FUNCTION_BLOCK FB_Afstandssensor IMPLEMENTS ITF_Afstandssensor
VAR_INPUT
END_VAR
VAR_OUTPUT
END_VAR
VAR
	// Interne waarden
	Afstand_Intern : LREAL;
	Drempelwaarde_Intern : LREAL;
	
	Detectie_Intern : BOOL;
	Status_Intern : E_AfstandssensorStatus;
END_VAR

PROPERTY Afstand : LREAL
GET
Afstand := Afstand_Intern;
END_GET
SET
VAR
	Waarde : LREAL;
END_VAR
Afstand_Intern := Waarde;
END_SET
END_PROPERTY

PROPERTY Detectie : BOOL
GET
Detectie := Detectie_Intern;
END_GET
END_PROPERTY

PROPERTY Drempelwaarde : LREAL
GET
Drempelwaarde := Drempelwaarde_Intern;
END_GET
SET
VAR
	Waarde : LREAL;
END_VAR
Drempelwaarde_Intern := Waarde;
END_SET
END_PROPERTY

PROPERTY Status : E_AfstandssensorStatus
GET
Status := Status_Intern;
END_GET
END_PROPERTY

METHOD Update : BOOL
// Afstandssensor controleert op interne fouten
IF Afstand_Intern < 0 THEN
	Status_Intern := E_AfstandssensorStatus.Error;
	Detectie_Intern := FALSE;
	RETURN;
END_IF

// Afstandssensor controleert op drempelwaarde
IF Afstand_Intern <= Drempelwaarde_Intern THEN
	Detectie_Intern := TRUE; 
	Status_Intern := E_AfstandssensorStatus.Detectie;
ELSE
	Detectie_Intern := FALSE; 
	Status_Intern := E_AfstandssensorStatus.Normaal;
END_IF
END_METHOD

END_FUNCTION_BLOCK

(* stored: Version 1.1.0.1
   POU FB_Afstandssensor: Id {72d78e64-2ca1-40bf-a72f-434aeebace35}, SpecialFunc None
   Folder Methods: Id {64d0ffcc-fbf0-4493-9adf-11821c75192c}
   Folder Properties: Id {55fd0682-a737-4488-9c0e-4e669ed9a091}
   Property Afstand: Id {3ecc7837-44c5-4438-ad48-9dbbd9fdfddd}
   Get Get: Id {096180e0-4b56-41a4-9b54-a7116699a87c}
   Set Set: Id {d6b94a18-1709-4e84-bd0b-bef362741fdc}
   Property Detectie: Id {a05856dd-e932-4ea4-a79e-b14c2d47b985}
   Get Get: Id {9d8828ce-fd1c-4e62-8d77-c8c2ea779023}
   Property Drempelwaarde: Id {c5ccdce1-5ede-45f5-8fcd-0e7ac99fca36}
   Get Get: Id {e4a41439-4cdd-46a5-8b96-572e91f496df}
   Set Set: Id {2dc47b39-e5b4-49c0-bb1b-99b78de7d685}
   Property Status: Id {dc749c30-2631-4802-ac58-41a05792b234}
   Get Get: Id {5aeacc10-aae3-4fe7-a989-8e248739e7bb}
   Method Update: Id {5deeb264-a5f9-4d49-9a81-a183613a6111} *)
